TYPE HydraulicsIOParts :
STRUCT
	///PG: Pumps Group
	pumpsGroup: HydraulicsPumpsGroupIO;
END_STRUCT
END_TYPE

(* stored: Version 1.1.0.1, ProductVersion 3.1.4019.2
   DUT HydraulicsIOParts: Id {57da5879-2be4-480b-a9ea-0212b33a2f4c} *)
